FUNCTION_BLOCK TestNodeFactory IMPLEMENTS ITF_NodeFactory
VAR
	CreatedCount : UDINT;
    DeletedCount : UDINT;
END_VAR

METHOD CreateNode : ITF_Node
VAR
	p : POINTER TO TestNode;
END_VAR
p := __NEW(TestNode);
IF p <> 0 THEN
    CreatedCount := CreatedCount + 1;
    CreateNode := p^;   // return as ITF_Node
END_IF
END_METHOD

METHOD DestroyNode : BOOL
VAR_INPUT
	Ptr	: PVOID;
END_VAR
VAR 
	p : POINTER TO TestNode; 
END_VAR
p := Ptr;
IF p <> 0 THEN
    __DELETE(p);
    DeletedCount := DeletedCount + 1;
    DestroyNode := TRUE;
END_IF
END_METHOD

METHOD DoesCreateEqualDestroy : BOOL
VAR_INPUT
END_VAR
IF CreatedCount = DeletedCount THEN

	DoesCreateEqualDestroy := TRUE;

ELSE

	DoesCreateEqualDestroy := FALSE;	

END_IF
END_METHOD

END_FUNCTION_BLOCK

(* stored: Version 1.1.0.1
   POU TestNodeFactory: Id {86dfbdba-ea10-4f54-a634-e4ef1602d238}, SpecialFunc None
   Method CreateNode: Id {e296f237-3883-49e8-b1f5-9aa807fd0b08}
   Method DestroyNode: Id {2134458c-6bdc-4c71-9dcf-e0fcb06b1cac}
   Method DoesCreateEqualDestroy: Id {61858ddc-b7b1-4c6e-847d-092222fb0e5f} *)
